FUNCTION Convert_DT_TO_TIME : Hresult
VAR_INPUT
	in : DT;
	out : REFERENCE TO TIME;
END_VAR
VAR
	converted : TIME;
END_VAR

converted := DT_TO_TIME(in);

IF (TIME_TO_DT(converted) <> in) THEN
	Convert_DT_TO_TIME := INCOMPATIBLE;
	RETURN;
END_IF

out := converted;

END_FUNCTION

(* stored: Version 1.1.0.1, ProductVersion 3.1.4024.12
   POU Convert_DT_TO_TIME: Id {1d768cac-a9e3-47a2-9222-b9361baa5b39}, SpecialFunc None *)
